# EPICS autosave request: softGlueApp/Db/GateDly_settings.req
$(P)$(H)GateDly-$(N)_CLK_Signal
$(P)$(H)GateDly-$(N)_IN_Signal
$(P)$(H)GateDly-$(N)_OUT_Signal
$(P)$(H)GateDly-$(N)_DLY
$(P)$(H)GateDly-$(N)_WIDTH
